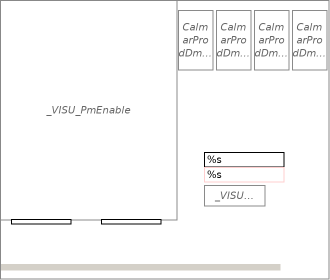
VISUALIZATION _VISU_Pm_WEU_mini  // 330x280
VAR_IN_OUT
  mInst : FB_PrintModule_WEU;
END_VAR
    Rectangle (0,0 330x280)
    Frame (204,185 61x21)
        shows _VISU_CameraTrigger(mInst := mInst.fbMarkDetection)
    Rectangle (204,152 80x15), "%s", tooltip "active camera device", text variable: mInst.fbWorkerCamera._iActiveCam.sName
    Rectangle (204,167 80x15), "%s", tooltip "active camera mode", text variable: mInst.fbWorkerCamera._iActiveCam.eCameraMode, colour toggle: mInst.fbWorkerCamera._bCamValid
    RoundedRectangle (0,264 280x6), colour toggle: mInst.fbView.bMovingInd
    Frame (0,0 177x220)
        shows _VISU_PmEnable(mInst := mInst)
        p2738717112: mInst.fbView.zPos_PM
    RoundedRectangle (11,219 60x5), colour toggle: mInst.fbView.bPrintInd[2]
        p2738717112: mInst.fbView.zPos_PM
    RoundedRectangle (101,219 60x5), colour toggle: mInst.fbView.bPrintInd[1]
        p2738717112: mInst.fbView.zPos_PM
    Line (0,0) (280,0)
    Frame (254,10 35x60)
        shows CalmarProdDmax._VISU_WorkerDefGrid_small(m_Inst := mInst.fbWorkerDeformation)
    Frame (292,10 35x60)
        shows CalmarProdDmax._VISU_WorkerDefGrid_small(m_Inst := mInst.fbWorkerCamera)
    Frame (178,10 35x60)
        shows CalmarProdDmax._VISU_WorkerDefGrid_small(m_Inst := mInst.fbWorkerPrint[2])
    Frame (216,10 35x60)
        shows CalmarProdDmax._VISU_WorkerDefGrid_small(m_Inst := mInst.fbWorkerPrint[1])
END_VISUALIZATION

(* stored: Version 1.1.0.1, ProductVersion 3.1.4024.11
   Visu _VISU_Pm_WEU_mini: Id {369d7b0f-c97e-4519-b200-3a08563d13af} *)
